(*
    This test-suite runs several asserts with the same parameters (same expected, actual, message), calling the asserts
    in different cycles and using the same test.
    On top of this, we will call new asserts (though with same parameters) in later cycles.
    The reason we want the framework to support this is that theoretically the user could want to do an assert with the
    same message, using the same test with the same data values for both expected and actual, and splitting the asserts
    on different cycles.
*)
{attribute 'call_after_init'}
FUNCTION_BLOCK FB_MultipleAssertWithSameParametersInDifferentCyclesAndInSameTest EXTENDS TcUnit.FB_TestSuite IMPLEMENTS TcUnit.I_RunnableTestSuite
VAR
    Assert : TcUnit.FB_Assert;
    TimerAgain : Tc2_Standard.TON := (PT := T#1S); // Timer to call "AssertSeveralTimesAgain"
    TimerAgainAgain : Tc2_Standard.TON := (PT := T#5S); // Timer to call "AssertSeveralTimesAgainAgain"
    CalledAll : BOOL; // Indication of whether we've called all tests
END_VAR

METHOD PRIVATE Assert_SeveralTimes
VAR
    a : DWORD := 16#12345678;
    b : DWORD := 16#90ABCDEF;

    c : DWORD := 16#12345678;
    d : DWORD := 16#90ABCDEF;

    e : DWORD := 16#12345678;
    f : DWORD := 16#90ABCDEF;
    
    g : DWORD := 16#12345678;
    h : DWORD := 16#90ABCDEF;
    
    i : DWORD := 16#12345678;
    j : DWORD := 16#90ABCDEF;
    
    k : DWORD := 16#12345678;
    l : DWORD := 16#90ABCDEF;
    
    m : DWORD := 16#12345678;
    n : DWORD := 16#90ABCDEF;
    
    o : DWORD := 16#12345678;
    p : DWORD := 16#90ABCDEF;
    
    q : DWORD := 16#12345678;
    rr : DWORD := 16#90ABCDEF;
END_VAR
TEST('Assert_SeveralTimes');

Assert.AssertEquals_DWORD(Expected := a,
                          Actual := b,
                          Message := 'Values differ');
Assert.AssertEquals_DWORD(Expected := c,
                          Actual := d,
                          Message := 'Values differ');
Assert.AssertEquals_DWORD(Expected := e,
                          Actual := f,
                          Message := 'Values differ');

TimerAgain(IN := TRUE);
IF TimerAgain.Q THEN
    TimerAgainAgain(IN := TRUE);
    Assert.AssertEquals_DWORD(Expected := g,
                              Actual := h,
                              Message := 'Values differ');
    Assert.AssertEquals_DWORD(Expected := i,
                              Actual := j,
                              Message := 'Values differ');
    Assert.AssertEquals_DWORD(Expected := k,
                              Actual := l,
                              Message := 'Values differ');
END_IF

IF TimerAgainAgain.Q THEN
    Assert.AssertEquals_DWORD(Expected := m,
                              Actual := n,
                              Message := 'Values differ');
    Assert.AssertEquals_DWORD(Expected := o,
                              Actual := p,
                              Message := 'Values differ');
    Assert.AssertEquals_DWORD(Expected := q,
                              Actual := rr,
                              Message := 'Values differ');
    CalledAll := TRUE;    
END_IF
END_METHOD

METHOD FB_init : BOOL
VAR_INPUT
	bInitRetains : BOOL; // if TRUE, the retain variables are initialized (warm start / cold start)
	bInCopyCode : BOOL;  // if TRUE, the instance afterwards gets moved into the copy code (online change)
END_VAR
SUPER^.RegisterTestSuite(THIS^);
END_METHOD

METHOD PUBLIC RunTests : TCUNIT.E_TestSuiteRunState
Assert_SeveralTimes();

IF CalledAll THEN
    RunTests := TCUNIT.E_TestSuiteRunState.FINISHED;
END_IF
END_METHOD

END_FUNCTION_BLOCK

(* stored: Version 1.1.0.1, ProductVersion 3.1.4022.16
   POU FB_MultipleAssertWithSameParametersInDifferentCyclesAndInSameTest: Id {b90749b6-04c8-4717-bf88-8db2fbf83f6a}, SpecialFunc None
   Method Assert_SeveralTimes: Id {fec25683-5d3d-4525-82ab-3bcd5de9b899}
   Method FB_init: Id {c346e23b-7954-4ef7-af50-5c27d0d11c81}
   Method RunTests: Id {f05b6079-4de6-4821-af92-17b216f18eeb} *)
